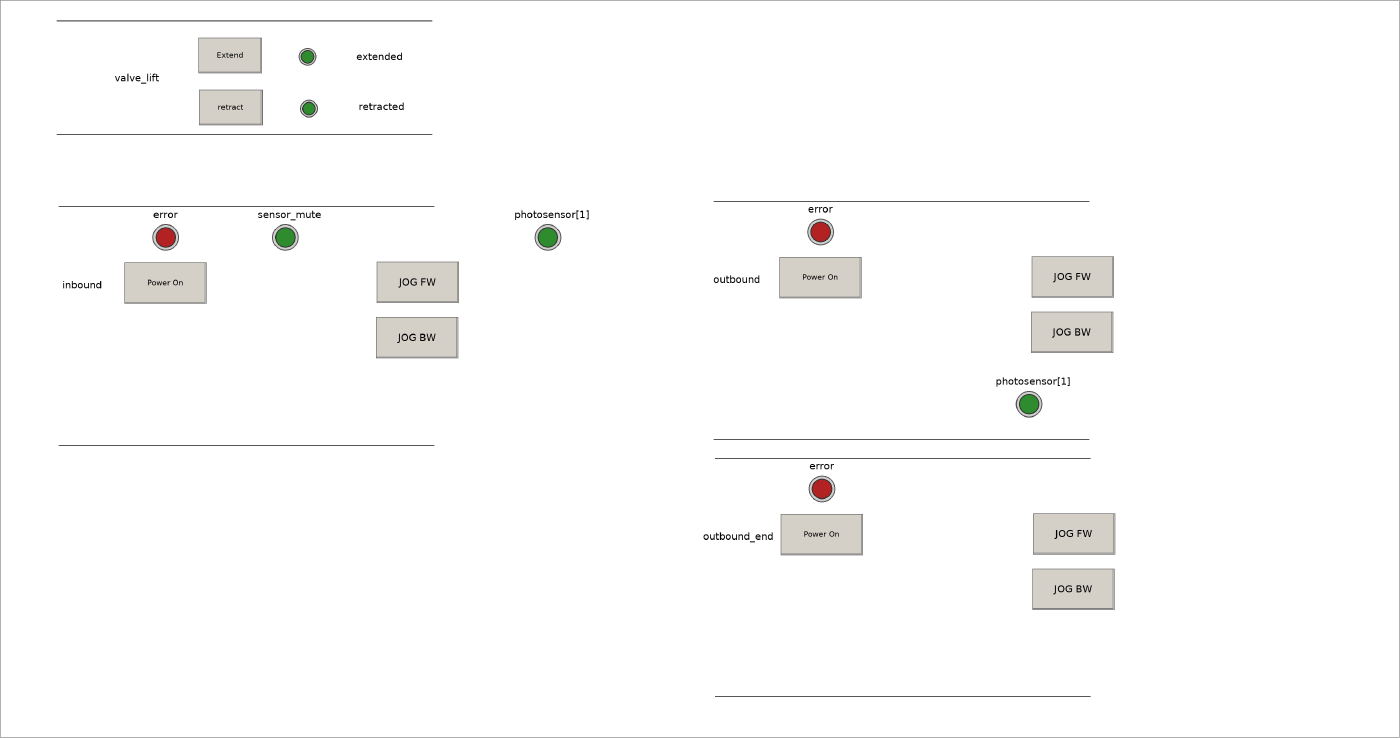
VISUALIZATION v_io_working  // 2048x1080
    Label (120,101 160x26), "valve_lift"
    Button (290,55 93x52), "Extend", colour toggle: GVL.fb_working.valve_lift.extend
        OnMouseDown: execute { GVL.fb_working.valve_lift.extend := TRUE; GVL.fb_working.valve_lift.retract := FALSE; }
    Button (291,131 93x52), "retract", colour toggle: GVL.fb_working.valve_lift.retract
        OnMouseDown: execute { GVL.fb_working.valve_lift.extend 	:= FALSE; GVL.fb_working.valve_lift.retract 	:= TRUE; }
    Lamp1 (435,68 30x30), variable: GVL.fb_working.valve_lift.extended, style: Lamp-Lamp1-Green
    Lamp1 (437,144 30x30), variable: GVL.fb_working.valve_lift.retracted, style: Lamp-Lamp1-Green
    Label (489,70 132x26), "extended"
    Label (492,143 132x26), "retracted"
    Line (83,196) (632,196)
    Line (83,30) (632,30)
    Lamp1 (220,325 45x45), variable: GVL.fb_working.roller_inbound.roller.err, style: Lamp-Lamp1-Red
    Label (176,301 132x26), "error"
    Line (86,302) (635,302)
    Button (551,383 120x60), "JOG FW", colour toggle: GVL.fb_working.roller_inbound.roller.forward
        OnMouseDown: execute { GVL.fb_working.roller_inbound.roller.forward	:= TRUE; }
        OnMouseUp: execute { GVL.fb_working.roller_inbound.roller.forward	:= FALSE; }
    Button (550,464 120x60), "JOG BW", colour toggle: GVL.fb_working.roller_inbound.roller.backward
        OnMouseDown: execute { GVL.fb_working.roller_inbound.roller.backward	:= TRUE; }
        OnMouseUp: execute { GVL.fb_working.roller_inbound.roller.backward	:= FALSE; }
    Button (182,384 120x60), "Power On", colour toggle: GVL.fb_working.roller_inbound.roller.Power
        toggle GVL.fb_working.roller_inbound.roller.Power
    Line (86,651) (635,651)
    Lamp1 (395,325 45x45), variable: GVL.fb_working.roller_inbound.photo_sensor_mute, style: Lamp-Lamp1-Green
    Label (351,301 145x26), "sensor_mute"
    Lamp1 (779,325 45x45), variable: GVL.fb_working.roller_inbound.photo_sensor, style: Lamp-Lamp1-Green
    Label (735,301 145x26), "photosensor[1]"
    Label (54,404 132x26), "inbound"
    Lamp1 (1178,317 45x45), variable: GVL.fb_working.roller_outbound.roller.err, style: Lamp-Lamp1-Red
    Label (1134,293 132x26), "error"
    Line (1044,294) (1593,294)
    Button (1509,375 120x60), "JOG FW", colour toggle: GVL.fb_working.roller_outbound.roller.forward
        OnMouseDown: execute { GVL.fb_working.roller_outbound.roller.forward	:= TRUE; }
        OnMouseUp: execute { GVL.fb_working.roller_outbound.roller.forward	:= FALSE; }
    Button (1508,456 120x60), "JOG BW", colour toggle: GVL.fb_working.roller_outbound.roller.backward
        OnMouseDown: execute { GVL.fb_working.roller_outbound.roller.backward	:= TRUE; }
        OnMouseUp: execute { GVL.fb_working.roller_outbound.roller.backward	:= FALSE; }
    Button (1140,376 120x60), "Power On", colour toggle: GVL.fb_working.roller_outbound.roller.Power
        toggle GVL.fb_working.roller_outbound.roller.Power
    Line (1044,643) (1593,643)
    Lamp1 (1483,569 45x45), variable: GVL.fb_working.roller_outbound.photo_sensor, style: Lamp-Lamp1-Green
    Label (1439,545 145x26), "photosensor[1]"
    Label (1012,396 132x26), "outbound"
    Lamp1 (1180,693 45x45), variable: GVL.fb_working.roller_outbound_end.roller.err, style: Lamp-Lamp1-Red
    Label (1136,669 132x26), "error"
    Line (1046,670) (1595,670)
    Button (1511,751 120x60), "JOG FW", colour toggle: GVL.fb_working.roller_outbound_end.roller.forward
        OnMouseDown: execute { GVL.fb_working.roller_outbound_end.roller.forward	:= TRUE; }
        OnMouseUp: execute { GVL.fb_working.roller_outbound_end.roller.forward	:= FALSE; }
    Button (1510,832 120x60), "JOG BW", colour toggle: GVL.fb_working.roller_outbound_end.roller.backward
        OnMouseDown: execute { GVL.fb_working.roller_outbound_end.roller.backward	:= TRUE; }
        OnMouseUp: execute { GVL.fb_working.roller_outbound_end.roller.backward	:= FALSE; }
    Button (1142,752 120x60), "Power On", colour toggle: GVL.fb_working.roller_outbound.roller.Power
        toggle GVL.fb_working.roller_outbound_end.roller.Power
    Line (1046,1019) (1595,1019)
    Label (1014,772 132x26), "outbound_end"
END_VISUALIZATION

(* stored: Version 1.1.0.1, ProductVersion 3.1.4024.12
   Visu v_io_working: Id {5c93d195-e8bd-46c5-b6cb-5d024bd76eab} *)
